Staubli VAL3: TRAJ.dtx

Trajectory tTraj
  [0]
    TrajectoryItem tSuper[3]
      [0]
        num distance
        num moveType = 1
        num nTime
        num nStop
        num nTcpAction
        string comment = "appro"
        bool toStop
        mdesc nom_speed = {tmax=300, rmax=9999, leave=30, reach=30}
        InstrItem iInstr[3]
          [0]
            string sType
            string sData
          [1]
            string sType
            string sData
          [2]
            string sType
            string sData
        num nMoveId
      [1]
        num distance = 2
        num moveType = 1
        num nTime
        num nStop
        num nTcpAction = 2
        string comment = "point"
        bool toStop = true
        mdesc nom_speed = {tmax=300, rmax=9999, leave=30, reach=30}
        InstrItem iInstr[3]
          [0]
            string sType
            string sData
          [1]
            string sType
            string sData
          [2]
            string sType
            string sData
        num nMoveId
      [2]
        num distance
        num moveType = 1
        num nTime
        num nStop
        num nTcpAction
        string comment = "depart"
        bool toStop
        mdesc nom_speed = {tmax=300, rmax=9999, leave=30, reach=30}
        InstrItem iInstr[3]
          [0]
            string sType
            string sData
          [1]
            string sType
            string sData
          [2]
            string sType
            string sData
        num nMoveId
    string sID = "POINT pose"
    num nId
public bool bMoveType[3]
  [0] = true
  [1] = true
  [2] = true
public bool bStepping
bool bToSave
frame fSetFrame = {fatherId=world[0]}
mdesc mMdesc = {accel=10, vel=10, decel=10, blend=off}
string sInstruction
public string sItems
string sMenu[8]
  [5] = "Duplicate"
  [7] = "New"
string sTrajType = "POINT"
pointRx pToGo[2]
  [0] = {fatherId=world[0]}
  [1] = {fatherId=world[0]}
num nFile
pointRx pPoints[3]
  [0] = {fatherId=world[0]}
  [1] = {fatherId=world[0]}
  [2] = {fatherId=world[0]}
Traies pEditPoint
  [0]
    frame fFrame
    num nIndexTool
    string sID
    num nIndexFrame
    TrajItem tData
      [0]
        TrajectoryItem tSuper
          [0]
            num distance
            num moveType
            num nTime
            num nStop
            num nTcpAction
            string comment
            bool toStop
            mdesc nom_speed = {tmax=300, rmax=9999, leave=30, reach=30}
            InstrItem iInstr[3]
              [0]
                string sType
                string sData
              [1]
                string sType
                string sData
              [2]
                string sType
                string sData
            num nMoveId
        pointRx pPoint
        num nType
        pointRx pCircle
string sTrajCycle
